(* CODESYS project slurryboss

Project tree, tasks and I/O mapping:
  CODESYS_Control_Win_V3_x64 : CODESYS Control Win V3 x64, CODESYS, version 3.5.20.0
    application Application
  CR1104 : ecomatDisplay43inch_64bit, ifm electronic, order no. 
      , version 3.5.19.4
    application Application
      libraries: ifmDevice_ecomatDisplay, * (ifm electronic); CmpBitmapPool, * (System); Util, 3.5.19.0 (System); Standard, 3.5.18.0 (System); SysTimer, * (System); BACnet2, 2.0.0.0 (CODESYS); CAA CiA 405, 4.1.0.0 (CAA Technical Workgroup); Element Collections, 3.5.17.0 (3S - Smart Software Solutions GmbH)
      task Task (cyclic, interval 1 ms, priority 0) calls PLC_PRG, Key_Lights, Test_PRG
      task VISU_TASK (cyclic, interval 10 ms, priority 15) calls VisuElems.Visu_Prg
      Components/
        KIQ Radar/
          function block fb_KIQ [LD]
          function block fbexample [LD]
        LMC500/
          data type eLMC500_State
          function block fb_LMC500 [LD]
        Purge/
          fb_Purge/
            data type ePurge_State
            function block fb_Purge [LD]: Volume_Calculation
            visualisation frame_PurgeStatus
        Slurry Pump/
          data type eSlurry_Pump_State
          function block fb_Slurry_Pump [LD]
        program Test_PRG [CFC]
        function block TOI [ST]
      Device/
        program Key_Lights [CFC]
      function block fb_KeyLight [ST]: Off, On, Set_Blue, Set_Green, Set_Previous, Set_Red, Set_White
      HMI/
        Components/
          Blind setting/
            visualisation f_BlindSetting
            function block fb_BlindSetting [LD]
          Buttons/
            visualisation f_Toggle_Button
          Checkbox/
            visualisation f_Checkbox
            function block fb_Checkbox [LD]
          Dial Indicator/
            visualisation f_DialIndicator
            function block fb_DialIndicator [ST]
          f_ProgressBar/
            visualisation f_ProgressBar
          global variables Global_Cards
          Menu/
            visualisation menu_demo
            image pool Menu_Images
            visualisation Menu_Item
            visualisation Right_Side_Nav
            function block swipe [LD]
          Pages/
            visualisation Analytics
            visualisation Chemistry
            visualisation Overview
            visualisation Pumps
            visualisation Purge
            visualisation Settings
          POUs/
            Hotkey/
              visualisation Tank_Frame
            function block Keypad_Navigation_FB [ST]: down, left, right, up
          interface selectable
          Setting Card/
            POUs/
              function block fb_Setting_Card [ST]: decrease, increase
            visualisation Test_Card
            Visus/
              visualisation Setting_Card_Frame
          visualisation Slurry_Pump_Card
      program PLC_PRG [CFC]
      global variables prvars
      program Test1 [CFC]
    Communication : Communication, ifm electronic, version 3.5.19.4
      CAN : CAN, ifm electronic, version 3.5.19.4
        CANbus_ecomatDisplay4_3 : CANbus_ecomatDisplay4.3, ifm electronic, version 1.0.0.0
          CANopen_Manager : CANopen_Manager, CODESYS, version 4.2.0.0
              settings: ConfigVersion = 50659584
            ODE3 : ODE3, Invertek Drives Ltd, order no. 0, version Revision=16#00000000, FileVersion=1.1, File=INVERTEK_ODE3_CANopen v3.00.eds
                settings: NODEIDSAVED = 1; SDO Timeout = 1000000; EXPERTSETTINGS = FALSE; Heartbeat-Producer Time = 200; Process by CANopenManager = TRUE; PDO 16#1401.COBID = 16#C0000301; Generic COBID = '$NODEID+16#C0000300'; Process by CANopenManager = TRUE; PDO 16#1800.Event Timer = 0; Process by CANopenManager = TRUE; PDO 16#1801.COBID = 16#C0000281; PDO 16#1801.Event Timer = 0; Generic COBID = '$NODEID+16#C0000280'; Process by CANopenManager = TRUE; Control Command Register.Subindex = 16#00; Speed Reference.Subindex = 16#00; User Ramp.Subindex = 16#00; no-name.Index = 16#0006; no-name.Subindex = 16#00; no-name.Index = 16#0006; no-name.Subindex = 16#00; no-name.Index = 16#0006; no-name.Subindex = 16#00; no-name.Index = 16#0006; no-name.Subindex = 16#00; no-name.Index = 16#0006; no-name.Subindex = 16#00; Drive Status Register.Subindex = 16#00; Motor Speed.Subindex = 16#00; Motor Current.Subindex = 16#00; Drive Temperature.Subindex = 16#00; DC Bus Voltage.Subindex = 16#00; Digital Input Status.Subindex = 16#00; Analog Input 1.Subindex = 16#00; Analog Input 2.Subindex = 16#00; SDO List.Set COB-ID sync.Index = 16#1005; SDO List.Set COB-ID sync.Subindex = 16#00; SDO List.Set COB-ID sync.Value = 16#00000080; SDO List.Set COB-ID sync.Size = 32; SDO List.Set COB-ID sync.AbortIfError = FALSE;
                  SDO List.Set COB-ID sync.JumpToLine = FALSE; SDO List.Set COB-ID sync.Line = 0; SDO List.Set Guardtime.Index = 16#100C; SDO List.Set Guardtime.Subindex = 16#00; SDO List.Set Guardtime.Value = 16#00000000; SDO List.Set Guardtime.Size = 16; SDO List.Set Guardtime.AbortIfError = FALSE; SDO List.Set Guardtime.JumpToLine = FALSE; SDO List.Set Guardtime.Line = 0; SDO List.Set Lifetime.Index = 16#100D; SDO List.Set Lifetime.Subindex = 16#00; SDO List.Set Lifetime.Value = 16#00000000; SDO List.Set Lifetime.Size = 8; SDO List.Set Lifetime.AbortIfError = FALSE; SDO List.Set Lifetime.JumpToLine = FALSE; SDO List.Set Lifetime.Line = 0; SDO List.Disable Emcy CobID.Index = 16#1014; SDO List.Disable Emcy CobID.Subindex = 16#00; SDO List.Disable Emcy CobID.Value = 16#80000081; SDO List.Disable Emcy CobID.Size = 32; SDO List.Disable Emcy CobID.AbortIfError = FALSE; SDO List.Disable Emcy CobID.JumpToLine = FALSE; SDO List.Disable Emcy CobID.Line = 0; SDO List.Set Emcy CobID.Index = 16#1014; SDO List.Set Emcy CobID.Subindex = 16#00; SDO List.Set Emcy CobID.Value = 16#00000081; SDO List.Set Emcy CobID.Size = 32; SDO List.Set Emcy CobID.AbortIfError = FALSE; SDO List.Set Emcy CobID.JumpToLine = FALSE; SDO List.Set Emcy CobID.Line = 0; SDO List.Set Heartbeat Producer.Index = 16#1017; SDO List.Set Heartbeat Producer.Subindex = 16#00; SDO List.Set Heartbeat Producer.Value = 16#000000C8; SDO List.Set Heartbeat Producer.Size = 16; SDO List.Set Heartbeat Producer.AbortIfError = FALSE; SDO List.Set Heartbeat Producer.JumpToLine = FALSE; SDO List.Set Heartbeat Producer.Line = 0; SDO List.Disable PDO.Index = 16#1400; SDO List.Disable PDO.Subindex = 16#01; SDO List.Disable PDO.Value = 16#C0000201;
                  SDO List.Disable PDO.Size = 32; SDO List.Disable PDO.AbortIfError = FALSE; SDO List.Disable PDO.JumpToLine = FALSE; SDO List.Disable PDO.Line = 0; SDO List.Set transmission type.Index = 16#1400; SDO List.Set transmission type.Subindex = 16#02; SDO List.Set transmission type.Value = 16#FE; SDO List.Set transmission type.Size = 8; SDO List.Set transmission type.AbortIfError = FALSE; SDO List.Set transmission type.JumpToLine = FALSE; SDO List.Set transmission type.Line = 0; SDO List.Clear pdo mapping.Index = 16#1600; SDO List.Clear pdo mapping.Subindex = 16#00; SDO List.Clear pdo mapping.Value = 16#0; SDO List.Clear pdo mapping.Size = 8; SDO List.Clear pdo mapping.AbortIfError = FALSE; SDO List.Clear pdo mapping.JumpToLine = FALSE; SDO List.Clear pdo mapping.Line = 0; SDO List.Set Mapping.Index = 16#1600; SDO List.Set Mapping.Subindex = 16#01; SDO List.Set Mapping.Value = 16#20000010; SDO List.Set Mapping.Size = 32; SDO List.Set Mapping.AbortIfError = FALSE; SDO List.Set Mapping.JumpToLine = FALSE; SDO List.Set Mapping.Line = 0; SDO List.Set Mapping.Index = 16#1600; SDO List.Set Mapping.Subindex = 16#02; SDO List.Set Mapping.Value = 16#20010010; SDO List.Set Mapping.Size = 32; SDO List.Set Mapping.AbortIfError = FALSE; SDO List.Set Mapping.JumpToLine = FALSE; SDO List.Set Mapping.Line = 0; SDO List.Set Mapping.Index = 16#1600; SDO List.Set Mapping.Subindex = 16#03; SDO List.Set Mapping.Value = 16#20030010; SDO List.Set Mapping.Size = 32; SDO List.Set Mapping.AbortIfError = FALSE; SDO List.Set Mapping.JumpToLine = FALSE; SDO List.Set Mapping.Line = 0; SDO List.Set Mapping.Index = 16#1600;
                  SDO List.Set Mapping.Subindex = 16#04; SDO List.Set Mapping.Value = 16#00060010; SDO List.Set Mapping.Size = 32; SDO List.Set Mapping.AbortIfError = FALSE; SDO List.Set Mapping.JumpToLine = FALSE; SDO List.Set Mapping.Line = 0; SDO List.Set number of mappings.Index = 16#1600; SDO List.Set number of mappings.Subindex = 16#00; SDO List.Set number of mappings.Value = 16#04; SDO List.Set number of mappings.Size = 8; SDO List.Set number of mappings.AbortIfError = FALSE; SDO List.Set number of mappings.JumpToLine = FALSE; SDO List.Set number of mappings.Line = 0; SDO List.Set and enable COB-ID.Index = 16#1400; SDO List.Set and enable COB-ID.Subindex = 16#01; SDO List.Set and enable COB-ID.Value = 16#40000201; SDO List.Set and enable COB-ID.Size = 32; SDO List.Set and enable COB-ID.AbortIfError = FALSE; SDO List.Set and enable COB-ID.JumpToLine = FALSE; SDO List.Set and enable COB-ID.Line = 0; SDO List.Disable PDO.Index = 16#1401; SDO List.Disable PDO.Subindex = 16#01; SDO List.Disable PDO.Value = 16#C0000301; SDO List.Disable PDO.Size = 32; SDO List.Disable PDO.AbortIfError = FALSE; SDO List.Disable PDO.JumpToLine = FALSE; SDO List.Disable PDO.Line = 0; SDO List.Disable PDO.Index = 16#1800; SDO List.Disable PDO.Subindex = 16#01; SDO List.Disable PDO.Value = 16#C0000181; SDO List.Disable PDO.Size = 32; SDO List.Disable PDO.AbortIfError = FALSE; SDO List.Disable PDO.JumpToLine = FALSE; SDO List.Disable PDO.Line = 0; SDO List.Set transmission type.Index = 16#1800; SDO List.Set transmission type.Subindex = 16#02; SDO List.Set transmission type.Value = 16#FE; SDO List.Set transmission type.Size = 8; SDO List.Set transmission type.AbortIfError = FALSE; SDO List.Set transmission type.JumpToLine = FALSE;
                  SDO List.Set transmission type.Line = 0; SDO List.Set inhibit time.Index = 16#1800; SDO List.Set inhibit time.Subindex = 16#03; SDO List.Set inhibit time.Value = 16#0000; SDO List.Set inhibit time.Size = 16; SDO List.Set inhibit time.AbortIfError = FALSE; SDO List.Set inhibit time.JumpToLine = FALSE; SDO List.Set inhibit time.Line = 0; SDO List.Clear pdo mapping.Index = 16#1A00; SDO List.Clear pdo mapping.Subindex = 16#00; SDO List.Clear pdo mapping.Value = 16#0; SDO List.Clear pdo mapping.Size = 8; SDO List.Clear pdo mapping.AbortIfError = FALSE; SDO List.Clear pdo mapping.JumpToLine = FALSE; SDO List.Clear pdo mapping.Line = 0; SDO List.Set Mapping.Index = 16#1A00; SDO List.Set Mapping.Subindex = 16#01; SDO List.Set Mapping.Value = 16#200A0010; SDO List.Set Mapping.Size = 32; SDO List.Set Mapping.AbortIfError = FALSE; SDO List.Set Mapping.JumpToLine = FALSE; SDO List.Set Mapping.Line = 0; SDO List.Set Mapping.Index = 16#1A00; SDO List.Set Mapping.Subindex = 16#02; SDO List.Set Mapping.Value = 16#200B0010; SDO List.Set Mapping.Size = 32; SDO List.Set Mapping.AbortIfError = FALSE; SDO List.Set Mapping.JumpToLine = FALSE; SDO List.Set Mapping.Line = 0; SDO List.Set Mapping.Index = 16#1A00; SDO List.Set Mapping.Subindex = 16#03; SDO List.Set Mapping.Value = 16#200D0010; SDO List.Set Mapping.Size = 32; SDO List.Set Mapping.AbortIfError = FALSE; SDO List.Set Mapping.JumpToLine = FALSE; SDO List.Set Mapping.Line = 0; SDO List.Set Mapping.Index = 16#1A00; SDO List.Set Mapping.Subindex = 16#04; SDO List.Set Mapping.Value = 16#20100010; SDO List.Set Mapping.Size = 32;
                  SDO List.Set Mapping.AbortIfError = FALSE; SDO List.Set Mapping.JumpToLine = FALSE; SDO List.Set Mapping.Line = 0; SDO List.Set number of mappings.Index = 16#1A00; SDO List.Set number of mappings.Subindex = 16#00; SDO List.Set number of mappings.Value = 16#04; SDO List.Set number of mappings.Size = 8; SDO List.Set number of mappings.AbortIfError = FALSE; SDO List.Set number of mappings.JumpToLine = FALSE; SDO List.Set number of mappings.Line = 0; SDO List.Set and enable COB-ID.Index = 16#1800; SDO List.Set and enable COB-ID.Subindex = 16#01; SDO List.Set and enable COB-ID.Value = 16#40000181; SDO List.Set and enable COB-ID.Size = 32; SDO List.Set and enable COB-ID.AbortIfError = FALSE; SDO List.Set and enable COB-ID.JumpToLine = FALSE; SDO List.Set and enable COB-ID.Line = 0; SDO List.Disable PDO.Index = 16#1801; SDO List.Disable PDO.Subindex = 16#01; SDO List.Disable PDO.Value = 16#C0000281; SDO List.Disable PDO.Size = 32; SDO List.Disable PDO.AbortIfError = FALSE; SDO List.Disable PDO.JumpToLine = FALSE; SDO List.Disable PDO.Line = 0; ConfigVersion = 50659584
                unmapped channels: Control Command Register, Speed Reference, User Ramp, no-name, Drive Status Register, Motor Speed, Motor Current, Drive Temperature
      Ethernet : Ethernet, ifm electronic, version 3.5.19.4
  5ce3da45-db07-42e7-a21c-a00fff4ed8f6|C:\Users\johnm\Downloads\Full-Circle-Icon.png
  5ce3da45-db07-42e7-a21c-a00fff4ed8f6|C:\Users\johnm\Pictures\analytics icon.png
  5ce3da45-db07-42e7-a21c-a00fff4ed8f6|C:\Users\johnm\Pictures\demo branding button.png
  5ce3da45-db07-42e7-a21c-a00fff4ed8f6|C:\Users\johnm\Pictures\pump_3815797.png
  5ce3da45-db07-42e7-a21c-a00fff4ed8f6|C:\Users\johnm\Pictures\pump inverted.png
  text list GlobalTextList
*)

// CR1104/Application/Components/LMC500/eLMC500_State
{attribute 'qualified_only'}
{attribute 'strict'}
TYPE eLMC500_State :
(
	Disconnected := 0,
	Faulted:= 10,
	No_Detection:= 20,
	Water_Detected:= 30
);
END_TYPE

// CR1104/Application/Components/Slurry Pump/eSlurry_Pump_State
{attribute 'strict'}
{attribute 'to_string'}
TYPE eSlurry_Pump_State :
(
	Off := 0, //initial pseudo-state
	Disabled:= 10,
	Stopped_HL:= 20,
	Stopped_LL:= 25,
	Standby:= 30,
	Running:= 40
);
END_TYPE

// CR1104/Application/Components/Purge/fb_Purge/ePurge_State

{attribute 'strict'}
{attribute 'to_string'}
TYPE ePurge_State :
(
	Off := 0, //initial pseudo-state. No state displayed
	Disabled:= 10, //disabled by operator
	Standby:= 20, //enabled, not purging
	Purging:= 30 //purging
);
END_TYPE

// CR1104/Application/prvars
{attribute 'qualified_only'}
VAR_GLOBAL PERSISTENT RETAIN
	purge_frequency: UINT; //purge after x gallons
	purge_duration: UINT;
	purge_enabled: BOOL;
	slurry_pump_enabled: BOOL;
END_VAR

// CR1104/Application/HMI/Components/Global_Cards
{attribute 'qualified_only'}
VAR_GLOBAL
	Test_Navigation_Selection: ARRAY [0..4, 0..4] OF BOOL;;
END_VAR

// CR1104/Application/PLC_PRG
PROGRAM PLC_PRG
VAR
	setkeys: ifmDevice.ResetKeyMapping;
	setleds: ifmDevice.SetKeyLED; 
	Brightness: UDINT:= 16#00999999;
END_VAR

setkeys(xExecute := TRUE); // ifmDevice.ResetKeyMapping
setleds(xEnable := TRUE, udiColour := Brightness); // ifmDevice.SetKeyLED

END_PROGRAM

// CR1104/Application/Device/Key_Lights
PROGRAM Key_Lights
VAR_INPUT
	Brightness: REAL:= 1;
END_VAR
VAR
	KL: ARRAY [0..5] OF fb_KeyLight;
	setleds: ifmDevice.SetKeyLED; 
	//LED: ifmDevice.ControlAllKeyLEDs;

END_VAR

(*
4 -> 0
2 -> 1
0 -> 2
5 -> 3
3 -> 4
1 -> 5
*)

KL[2](Brightness_Setting := Brightness); // fb_KeyLight
KL[3](Brightness_Setting := Brightness); // fb_KeyLight
KL[1](Brightness_Setting := Brightness); // fb_KeyLight
KL[4](Brightness_Setting := Brightness); // fb_KeyLight
KL[0](Brightness_Setting := Brightness); // fb_KeyLight
KL[5](Brightness_Setting := Brightness); // fb_KeyLight
setleds(
    xEnable := NOT(setleds.xError),
    eLED_ID := ifmDevice.eKEY_LED_ID.KEY2_NAVIGATION,
    udiColour := KL[2].Color); // ifmDevice.SetKeyLED

END_PROGRAM

// CR1104/Application/fb_KeyLight
FUNCTION_BLOCK fb_KeyLight
VAR_INPUT
	Brightness_Setting: REAL:= 1; //0..1 real factor
END_VAR
VAR_OUTPUT
	Color: UDINT;
END_VAR
VAR
//	LED: ifmDevice.keyled;
	Red: REAL;
	Green: REAL;
	Blue: REAL;
	Light: REAL;
	Color_Memory: ARRAY [0..1] OF UDINT;
END_VAR

Color:=(
	SHL(TO_UDINT(Red * Light),16) + 	//16#00FF0000 values
	SHL(TO_UDINT(Green * Light),8) + 	//16#0000FF00 values
	TO_UDINT(Blue * Light)				//16#000000FF
);

IF Color_Memory[1] <> Color THEN
	Color_Memory[0]:= Color_Memory[1];
	Color_Memory[1]:= Color;
END_IF

METHOD Off
VAR_INPUT
END_VAR
THIS^.Light:= 0;
END_METHOD

METHOD On
VAR_INPUT
END_VAR
THIS^.Light:= THIS^.Brightness_Setting;
END_METHOD

METHOD Set_Blue
VAR_INPUT
END_VAR
THIS^.Red:= 0;
THIS^.Green:= 0;
THIS^.Blue:= 255;
END_METHOD

METHOD Set_Green
VAR_INPUT
END_VAR
END_METHOD

METHOD Set_Previous
VAR_INPUT
END_VAR
Red:= 	TO_REAL(16#00FF0000 AND Color_Memory[0]);
Green:= TO_REAL(16#0000FF00 AND Color_Memory[0]);
Blue:= 	TO_REAL(16#000000FF AND Color_Memory[0]);
END_METHOD

METHOD Set_Red
VAR_INPUT
END_VAR
END_METHOD

METHOD Set_White
VAR_INPUT
END_VAR
THIS^.Red:= 255;
THIS^.Green:= 255;
THIS^.Blue:= 255;
END_METHOD

END_FUNCTION_BLOCK

// CR1104/Application/Components/Test_PRG
PROGRAM Test_PRG
/////
VAR
	Purge_Control: fb_Purge;
	Slurry_Pump_Control: fb_Slurry_Pump;
	Slurry_Sensor: fb_LMC500;
	placeholder: ifmDevice.stKEY_MAP_LIST:= (eKey2_Return:= ifmDevice.eKey_Map_Codes.END);
	test_bit: BOOL;
END_VAR
/////
VAR
	Simu_Sys_On: BOOL;
	Simu_Pump_State: eSlurry_Pump_State;
	Simu_Tank_Level: UINT; 
	Simu_Sensor: eLMC500_State:= eLMC500_State.Water_Detected;
	keymap: ifmdevice.GetKeyMapping;
	set_map: ifmdevice.SetKeyMapping;
	test_toggle: fb_Checkbox;
	menu_swipe: swipe;
	Swipe_menu: BOOL;
END_VAR
/////

Slurry_Pump_Control(
    System_On := TRUE,
    Enabled := prvars.slurry_pump_enabled,
    Sensor := simu_sensor,
    Tank_Level := Simu_Tank_Level,
    Delay_Time := T#20s); // fb_Slurry_Pump
Purge_Control(
    System_On := TRUE,
    Enabled := prvars.purge_enabled,
    Pump_State := Slurry_Pump_Control.State,
    Gallons_Setpoint := prvars.purge_frequency,
    Purge_Duration := TO_TIME(prvars.purge_duration * 1000)); // fb_Purge
keymap(xExecute := NOT(keymap.xDone) AND NOT(keymap.xDone)); // ifmdevice.GetKeyMapping
set_map(xExecute := NOT(set_map.xDone OR set_map.xError), stKeyMapList := placeholder); // ifmdevice.SetKeyMapping
// parameter Slurry_Sensor.No_Detection_Value := 80
// parameter Slurry_Sensor.Detection_Value := 60
Slurry_Sensor(); // fb_LMC500
test_toggle(on := prvars.purge_enabled); // fb_Checkbox
// parameter menu_swipe.delay := T#1ms
// parameter menu_swipe.distance := 126
menu_swipe(on := Swipe_menu); // swipe
// TO_UINT(TO_REAL((Test_PRG.Purge_Control.Cycle_Volume) / TO_REAL(Test_PRG.Purge_Control.Gallons_Setpoint)) * 100): input not connected

END_PROGRAM

// CR1104/Application/Components/Purge/fb_Purge/fb_Purge
FUNCTION_BLOCK fb_Purge
VAR_INPUT
	System_On: BOOL;
	Enabled: BOOL;
	Hand_Purge: BOOL;
	Pump_State: eSlurry_Pump_State;
	Gallons_Setpoint: UINT; //how many gallons from ref_Slurry_Pump before purging
	Purge_Duration: TIME;
END_VAR
VAR_INPUT CONSTANT
	Time_To_Gallons: UINT:= 666; //ms per gallon
END_VAR
VAR_OUTPUT
	State: ePurge_State;
	Cycle_Volume: UINT;
END_VAR
VAR
	tmr_purge: TON;
	Cycle_Timer: TOI;
	ft_purge: F_TRIG;
END_VAR
VAR // added by the converter: edge detectors and wires of the graphical bodies
    _w1, _w2, _w3, _w4, _w5 : BOOL;
END_VAR

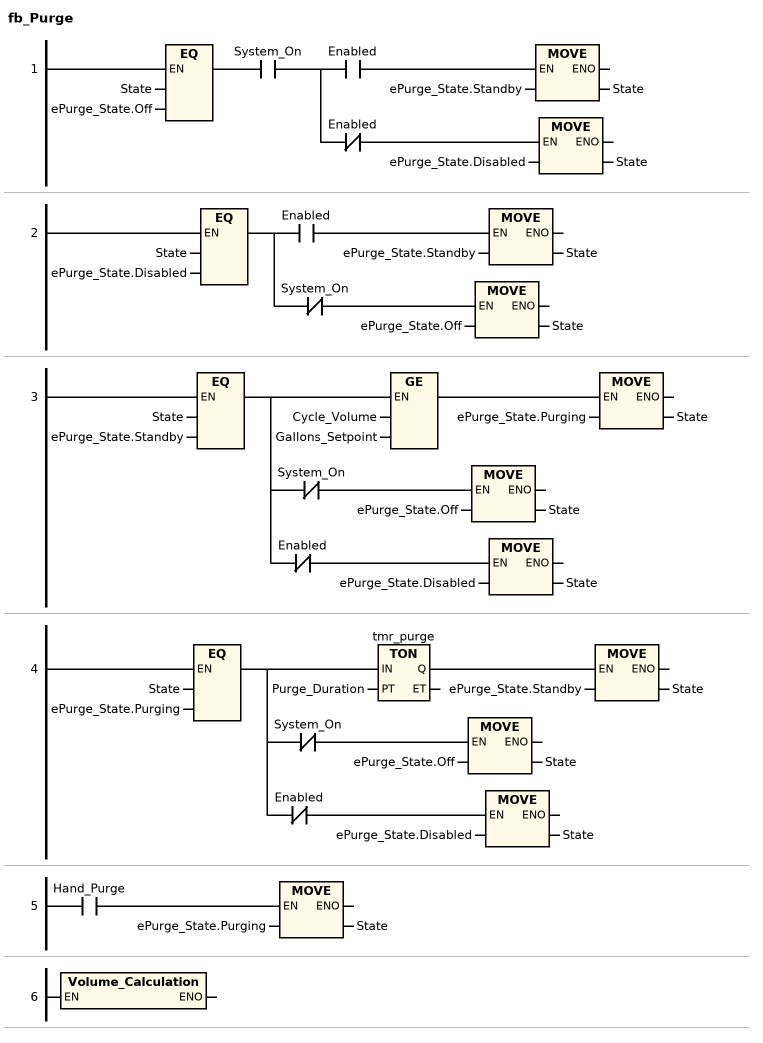
// NETWORK 1
_w1 := State = ePurge_State.Off AND System_On;
IF _w1 AND Enabled THEN State := ePurge_State.Standby; END_IF
IF _w1 AND NOT Enabled THEN State := ePurge_State.Disabled; END_IF

// NETWORK 2
_w2 := State = ePurge_State.Disabled;
IF _w2 AND Enabled THEN State := ePurge_State.Standby; END_IF
IF _w2 AND NOT System_On THEN State := ePurge_State.Off; END_IF

// NETWORK 3
_w3 := State = ePurge_State.Standby;
IF _w3 AND Cycle_Volume >= Gallons_Setpoint THEN State := ePurge_State.Purging; END_IF
IF _w3 AND NOT System_On THEN State := ePurge_State.Off; END_IF
IF _w3 AND NOT Enabled THEN State := ePurge_State.Disabled; END_IF

// NETWORK 4
_w4 := State = ePurge_State.Purging;
tmr_purge(IN := _w4, PT := Purge_Duration); // TON
IF tmr_purge.Q THEN State := ePurge_State.Standby; END_IF
IF _w4 AND NOT System_On THEN State := ePurge_State.Off; END_IF
IF _w4 AND NOT Enabled THEN State := ePurge_State.Disabled; END_IF

// NETWORK 5
IF Hand_Purge THEN State := ePurge_State.Purging; END_IF

// NETWORK 6
Volume_Calculation();

ACTION Volume_Calculation:
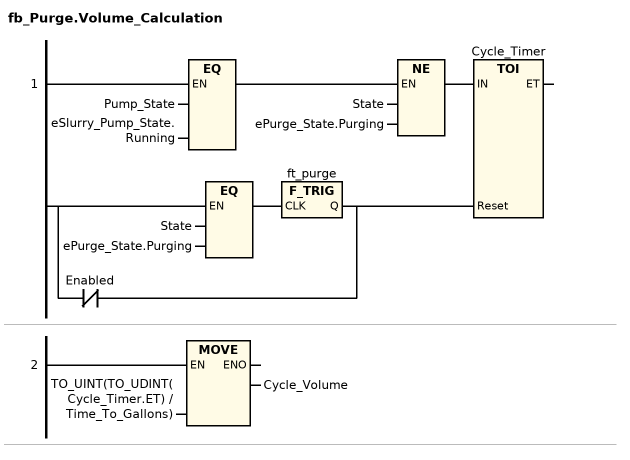
// NETWORK 1
_w5 := NOT Enabled;
IF NOT _w5 THEN
    ft_purge(CLK := State = ePurge_State.Purging); // F_TRIG
    _w5 := ft_purge.Q;
END_IF
Cycle_Timer(IN := Pump_State = eSlurry_Pump_State.Running AND State <> ePurge_State.Purging, Reset := _w5); // TOI

// NETWORK 2
Cycle_Volume := TO_UINT(TO_UDINT(Cycle_Timer.ET) / Time_To_Gallons);
END_ACTION

END_FUNCTION_BLOCK

// CR1104/Application/Components/TOI
FUNCTION_BLOCK TOI
VAR_INPUT
	IN : BOOL;
	Reset : BOOL;
END_VAR
VAR 
	TimerAdd: TIME; 
	CountingTimer: TIME;
	Trig: BOOL; 
	History: BOOL; 
	Pulse: BOOL; 
	TimerReset: BOOL; 
	Run: BOOL; 
	Running: BOOL; 
	StartTime: TIME;
	ResetONS: R_TRIG;
 END_VAR
 VAR_OUTPUT
	ET: TIME;
 END_VAR

ET:= TimerAdd + CountingTimer;
IF NOT IN THEN 
	IF Trig AND NOT History THEN 
		Pulse:= 1; History:= 1; Trig:= 0;
		ELSE 
			Pulse:= 0; History:= 1;
	END_IF
	IF Pulse THEN 
		CountingTimer:= ET;
	END_IF
	TimerReset:= 1;
END_IF
IF IN THEN 
	TimerReset:= 0;
	Trig:= 1; History:= 00;
END_IF
IF Reset THEN 
	TimerReset:= 1;
	CountingTimer:= T#001MS;
	ET:= T#001MS;
END_IF

Run:= NOT(TimerReset);

IF Run AND NOT Running THEN
	StartTime:= TIME();
	Running:= TRUE; END_IF
IF NOT Run AND NOT Running THEN
	StartTime:= TIME(); END_IF
ResetONS(clk:= TimerReset); 
IF ResetONS.Q THEN
	Running:= FALSE;
	StartTime:= TIME(); 
END_IF

TimerAdd:= TIME()-StartTime;

END_FUNCTION_BLOCK

// CR1104/Application/Components/Slurry Pump/fb_Slurry_Pump
FUNCTION_BLOCK fb_Slurry_Pump
VAR_INPUT
	System_On: BOOL;
	Enabled: BOOL;
	Sensor: eLMC500_State;
	Tank_Level: UINT;
	Delay_Time: TIME;
END_VAR
VAR_OUTPUT
	State: eSlurry_Pump_State;
END_VAR
VAR
	tmr_delay: TON;
	tmr_off: TON;
END_VAR
VAR // added by the converter: edge detectors and wires of the graphical bodies
    _w1, _w2, _w3, _w4, _w5 : BOOL;
END_VAR

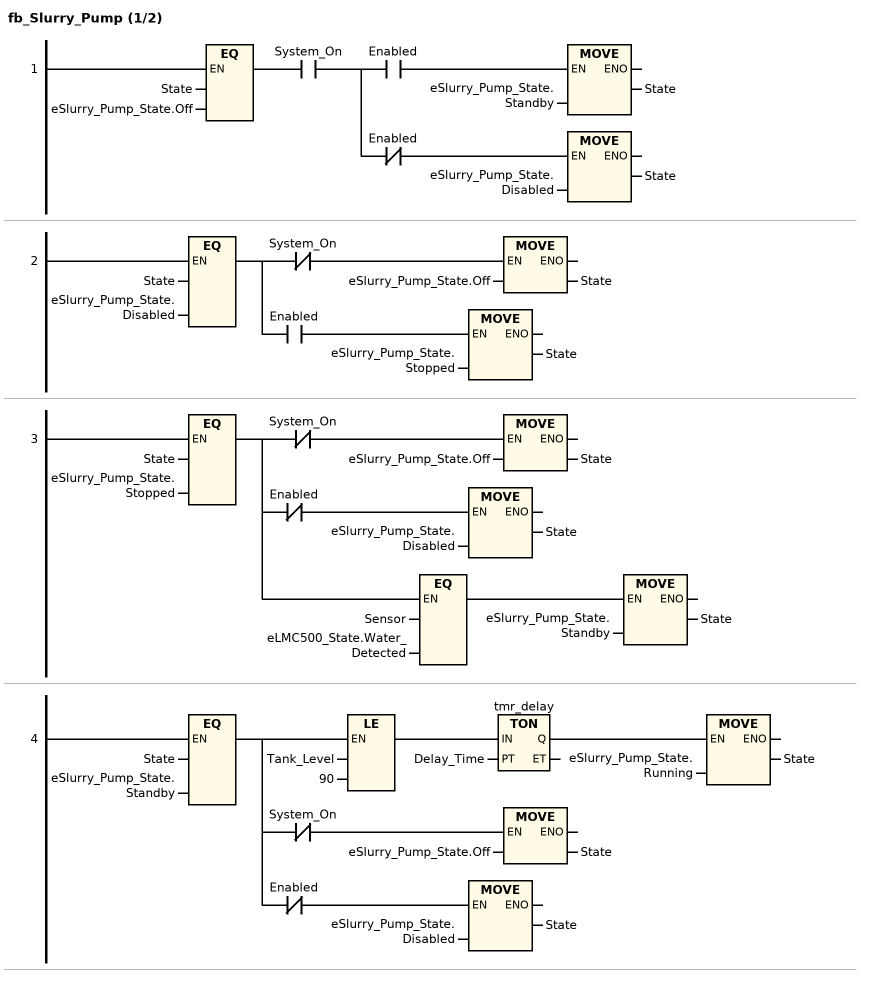
// NETWORK 1
_w1 := State = eSlurry_Pump_State.Off AND System_On;
IF _w1 AND Enabled THEN State := eSlurry_Pump_State.Standby; END_IF
IF _w1 AND NOT Enabled THEN State := eSlurry_Pump_State.Disabled; END_IF

// NETWORK 2
_w2 := State = eSlurry_Pump_State.Disabled;
IF _w2 AND NOT System_On THEN State := eSlurry_Pump_State.Off; END_IF
IF _w2 AND Enabled THEN State := eSlurry_Pump_State.Stopped; END_IF

// NETWORK 3
_w3 := State = eSlurry_Pump_State.Stopped;
IF _w3 AND NOT System_On THEN State := eSlurry_Pump_State.Off; END_IF
IF _w3 AND NOT Enabled THEN State := eSlurry_Pump_State.Disabled; END_IF
IF _w3 AND Sensor = eLMC500_State.Water_Detected THEN State := eSlurry_Pump_State.Standby; END_IF

// NETWORK 4
_w4 := State = eSlurry_Pump_State.Standby;
tmr_delay(IN := _w4 AND Tank_Level <= 90, PT := Delay_Time); // TON
IF tmr_delay.Q THEN State := eSlurry_Pump_State.Running; END_IF
IF _w4 AND NOT System_On THEN State := eSlurry_Pump_State.Off; END_IF
IF _w4 AND NOT Enabled THEN State := eSlurry_Pump_State.Disabled; END_IF

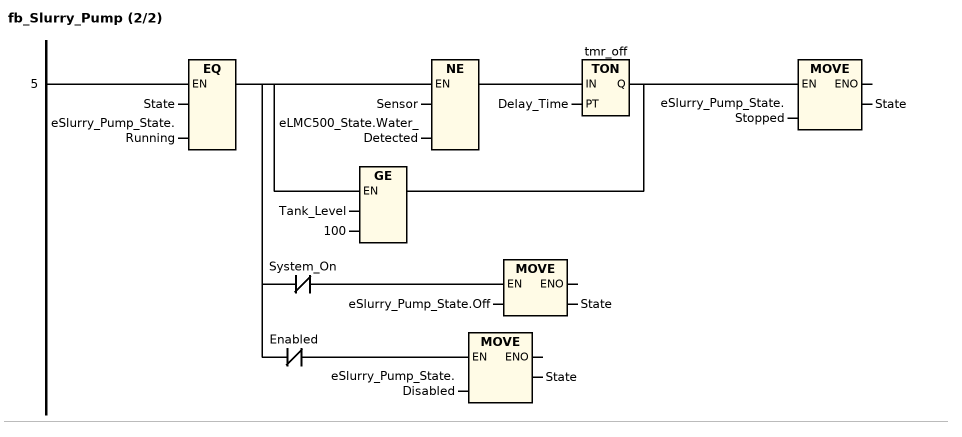
// NETWORK 5
_w5 := State = eSlurry_Pump_State.Running;
tmr_off(IN := _w5 AND Sensor <> eLMC500_State.Water_Detected, PT := Delay_Time); // TON
IF tmr_off.Q OR _w5 AND Tank_Level >= 100 THEN State := eSlurry_Pump_State.Stopped; END_IF
IF _w5 AND NOT System_On THEN State := eSlurry_Pump_State.Off; END_IF
IF _w5 AND NOT Enabled THEN State := eSlurry_Pump_State.Disabled; END_IF

END_FUNCTION_BLOCK

// CR1104/Application/Components/LMC500/fb_LMC500
FUNCTION_BLOCK fb_LMC500
/// 
VAR_INPUT
	IOL_Read: ARRAY [0..7] OF WORD;
END_VAR
///
VAR_OUTPUT
	state: eLMC500_State;
END_VAR
///
VAR_INPUT CONSTANT
	Detection_Value: UINT; //0-100
	No_Detection_Value: UINT; //0-100
END_VAR

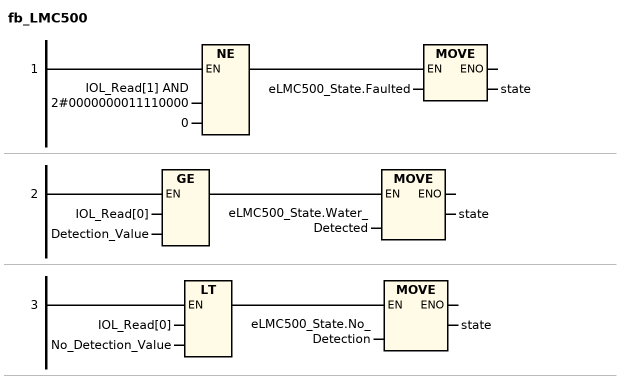
// NETWORK 1
IF (IOL_Read[1] AND 2#0000000011110000) <> 0 THEN state := eLMC500_State.Faulted; END_IF

// NETWORK 2
IF IOL_Read[0] >= Detection_Value THEN state := eLMC500_State.Water_Detected; END_IF

// NETWORK 3
IF IOL_Read[0] < No_Detection_Value THEN state := eLMC500_State.No_Detection; END_IF

END_FUNCTION_BLOCK

// CR1104/Application/HMI/Components/Checkbox/fb_Checkbox
FUNCTION_BLOCK fb_Checkbox
/////
VAR_IN_OUT
	on: BOOL;
END_VAR
/////
VAR_OUTPUT
	position: UINT;
END_VAR
////
VAR
	pos_ctu: CTU;
	pos_ctd: CTD;
	tmr_delay: TON;
	tmr_delay2: TON;
	off_trig: R_TRIG;
END_VAR
/////
VAR_INPUT CONSTANT
	delay: TIME:= T#2MS;
END_VAR
/////

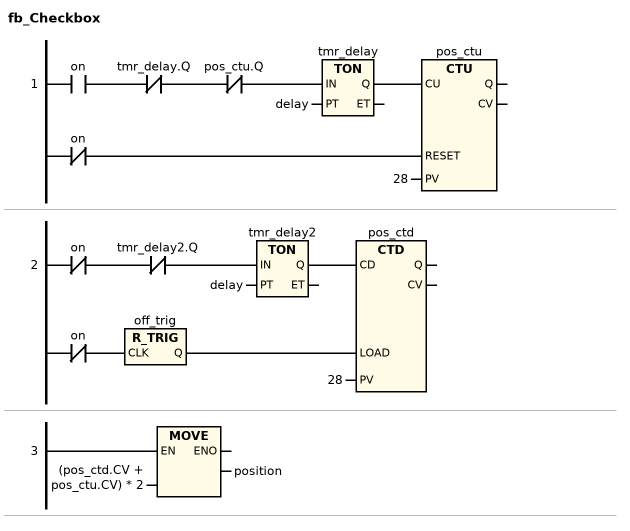
// NETWORK 1
tmr_delay(IN := on AND NOT tmr_delay.Q AND NOT pos_ctu.Q, PT := delay); // TON
pos_ctu(CU := tmr_delay.Q, RESET := NOT on, PV := 28); // CTU

// NETWORK 2
tmr_delay2(IN := NOT on AND NOT tmr_delay2.Q, PT := delay); // TON
off_trig(CLK := NOT on); // R_TRIG
pos_ctd(CD := tmr_delay2.Q, LOAD := off_trig.Q, PV := 28); // CTD

// NETWORK 3
position := (pos_ctd.CV + pos_ctu.CV) * 2;

END_FUNCTION_BLOCK

// CR1104/Application/HMI/Components/Menu/swipe
FUNCTION_BLOCK swipe
VAR_INPUT
	on: BOOL;
END_VAR
VAR_OUTPUT
	position: UINT;
END_VAR
VAR
	pos_ctu: CTU;
	pos_ctd: CTD;
	tmr_delay: TON;
	tmr_delay2: TON;
	off_trig: R_TRIG;
END_VAR
VAR_INPUT CONSTANT
	delay: TIME:= T#2MS;
	distance: UINT;
END_VAR

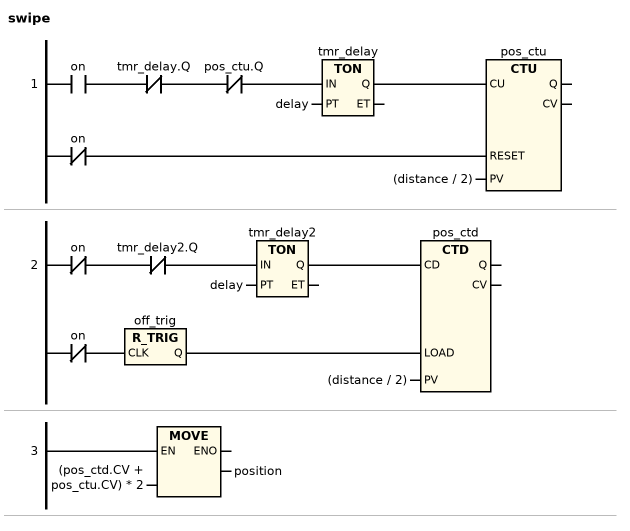
// NETWORK 1
tmr_delay(IN := on AND NOT tmr_delay.Q AND NOT pos_ctu.Q, PT := delay); // TON
pos_ctu(CU := tmr_delay.Q, RESET := NOT on, PV := (distance / 2)); // CTU

// NETWORK 2
tmr_delay2(IN := NOT on AND NOT tmr_delay2.Q, PT := delay); // TON
off_trig(CLK := NOT on); // R_TRIG
pos_ctd(CD := tmr_delay2.Q, LOAD := off_trig.Q, PV := (distance / 2)); // CTD

// NETWORK 3
position := (pos_ctd.CV + pos_ctu.CV) * 2;

END_FUNCTION_BLOCK

// CR1104/Application/Test1
PROGRAM Test1
VAR //test
END_VAR

END_PROGRAM

// CR1104/Application/Components/KIQ Radar/fb_KIQ
FUNCTION_BLOCK fb_KIQ
VAR_INPUT
END_VAR
VAR_OUTPUT
END_VAR
VAR
END_VAR

// NETWORK 1

END_FUNCTION_BLOCK

// CR1104/Application/Components/KIQ Radar/fbexample
FUNCTION_BLOCK fbexample
VAR_INPUT
END_VAR
VAR_OUTPUT
END_VAR
VAR
	active: BOOL;
	start_s2: BOOL;
	valve_q1: BOOL;
	highlevel_s5: BOOL;
	manual: BOOL;
	manual_mode: BOOL;
	manual_q1_button: BOOL;
END_VAR

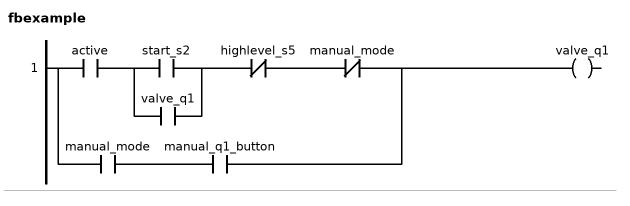
// NETWORK 1
valve_q1 := active AND (start_s2 OR valve_q1) AND NOT highlevel_s5 AND NOT manual_mode OR manual_mode AND manual_q1_button;

END_FUNCTION_BLOCK

// CR1104/Application/HMI/Components/selectable
INTERFACE selectable

END_INTERFACE

// CR1104/Application/HMI/Components/Blind setting/fb_BlindSetting
FUNCTION_BLOCK fb_BlindSetting
VAR_INPUT
	hover: BOOL;
	select: BOOL;
END_VAR
VAR_OUTPUT
	position: UINT;
END_VAR
VAR
	swipe_open: swipe;
END_VAR

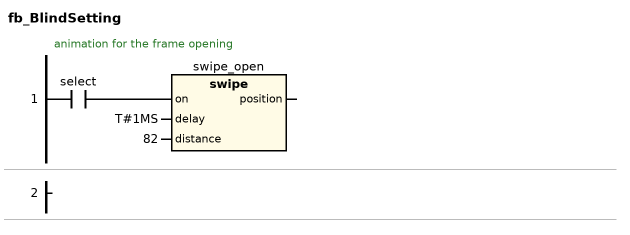
// NETWORK 1
// animation for the frame opening
swipe_open(on := select, delay := T#1MS, distance := 82); // swipe

// NETWORK 2

END_FUNCTION_BLOCK

// CR1104/Application/HMI/Components/Dial Indicator/fb_DialIndicator
FUNCTION_BLOCK fb_DialIndicator
VAR_INPUT
	r_Value: REFERENCE TO REAL;
	ui_Value: REFERENCE TO UINT;
	t_Value: REFERENCE TO TIME;
	Max_Value: UINT; //ms for time
	Name: STRING;
	Units: STRING;
END_VAR
VAR_OUTPUT
	Indicator_Val: UINT;
	xREAL: BOOL;
	xUINT: BOOL;
	xTIME: BOOL;
END_VAR
VAR
END_VAR


xREAL:= __ISVALIDREF(r_Value);
xUINT:= __ISVALIDREF(ui_Value);
xTIME:= __ISVALIDREF(t_Value);

IF xREAL THEN
	Indicator_Val:= 180 - TO_UINT((r_Value / TO_REAL(Max_Value)) * 180.0); //coefficient from proportion of max val
END_IF

END_FUNCTION_BLOCK

// CR1104/Application/HMI/Components/POUs/Keypad_Navigation_FB
FUNCTION_BLOCK Keypad_Navigation_FB
VAR_INPUT CONSTANT
	X_items: USINT; // How many items wide is the selection
	Y_items: USINT; // How many items tall is the selection
END_VAR
VAR_OUTPUT
	Position_X: USINT:= 0; //starting spot x
	Position_Y: USINT:= 0; //starting spot y
END_VAR

METHOD down
IF THIS^.Position_Y < THIS^.Y_items - 1 THEN
	THIS^.Position_Y:= THIS^.Position_Y + 1;
END_IF
END_METHOD

METHOD left
VAR_INPUT
END_VAR
IF THIS^.Position_X > 0 THEN
	THIS^.Position_X := THIS^.Position_X - 1;
END_IF
END_METHOD

METHOD right
VAR_INPUT
END_VAR
IF THIS^.Position_X < THIS^.X_Items - 1 THEN
	THIS^.Position_X := THIS^.Position_X + 1;
END_IF
END_METHOD

METHOD up
VAR_INPUT
END_VAR
IF THIS^.Position_Y > 0 THEN
	THIS^.Position_Y:= THIS^.Position_Y - 1;
END_IF
END_METHOD

END_FUNCTION_BLOCK

// CR1104/Application/HMI/Components/Setting Card/POUs/fb_Setting_Card
FUNCTION_BLOCK fb_Setting_Card
VAR_IN_OUT
	Value: UINT;
END_VAR
VAR_INPUT
	increment: UINT:= 1;
END_VAR
VAR_INPUT CONSTANT
	maximum: UINT;
	minimum: UINT;
END_VAR
VAR_OUTPUT
END_VAR
VAR
END_VAR

METHOD decrease
VAR_INPUT
END_VAR
IF THIS^.minimum >= THIS^.Value THEN
	RETURN;
END_IF

THIS^.Value:= THIS^.Value - increment;
END_METHOD

METHOD increase
VAR_INPUT
END_VAR
IF THIS^.maximum <= THIS^.Value THEN
	RETURN;
END_IF

THIS^.Value:= THIS^.Value + increment;
END_METHOD

END_FUNCTION_BLOCK

// CR1104/Application/HMI/Components/Slurry_Pump_Card
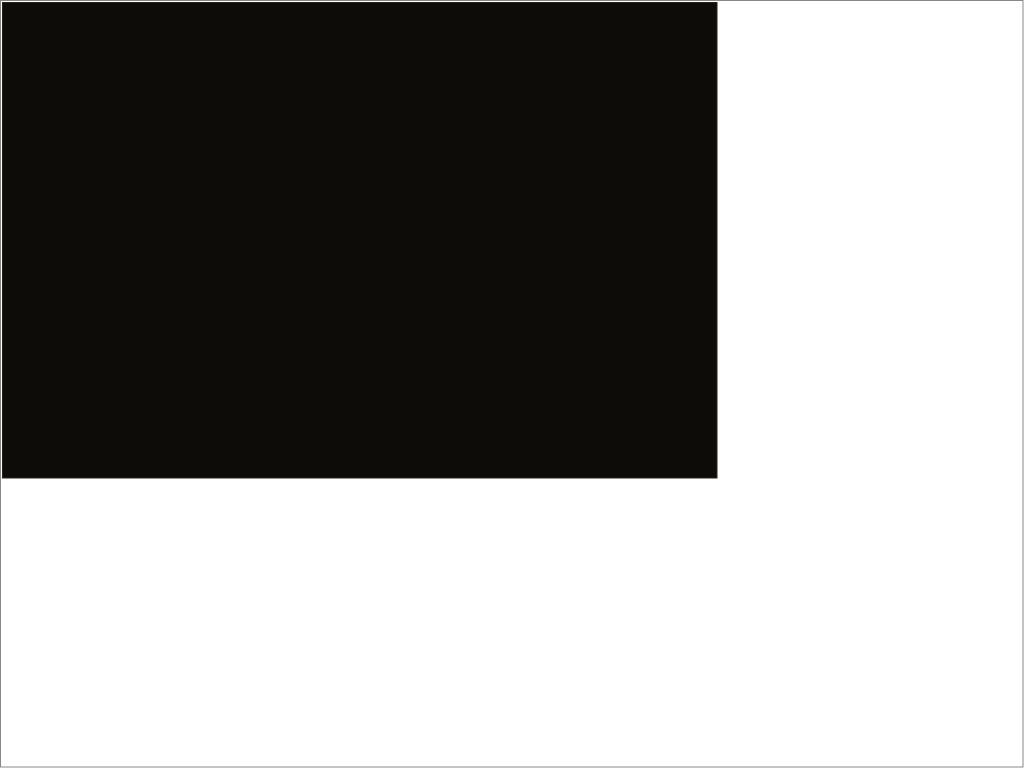
VISUALIZATION Slurry_Pump_Card  // 1024x768
VAR_INPUT
	_SELECTED: BOOL;
END_VAR
VAR
	Navigate: Keypad_Navigation_FB; 
END_VAR
    RoundedRectangle (2,2 715x476), colour toggle: _SELECTED
        p3560616238: TO_INT(_SELECTED) * (-116)
    hotkey  Id=481040531456, Key=KeyDown=True, KeyName=up, ActionToExecute=Action=STSnippet=IF NOT(_SELECTED) THEN RETURN; END_IF Navigate.up();, VisuElemId=-1
    hotkey  Id=481039482880, Key=KeyDown=True, KeyName=down, ActionToExecute=Action=STSnippet=IF NOT(_SELECTED) THEN RETURN; END_IF Navigate.down();, VisuElemId=-1
    hotkey  Id=481038434304, Key=KeyDown=True, KeyName=left, ActionToExecute=Action=STSnippet=IF NOT(_SELECTED) THEN RETURN; END_IF Navigate.left();, VisuElemId=-1
    hotkey  Id=481037385728, Key=KeyDown=True, KeyName=right, ActionToExecute=Action=STSnippet=IF NOT(_SELECTED) THEN RETURN; END_IF Navigate.right();, VisuElemId=-1
END_VISUALIZATION

// CR1104/Application/Components/Purge/fb_Purge/frame_PurgeStatus
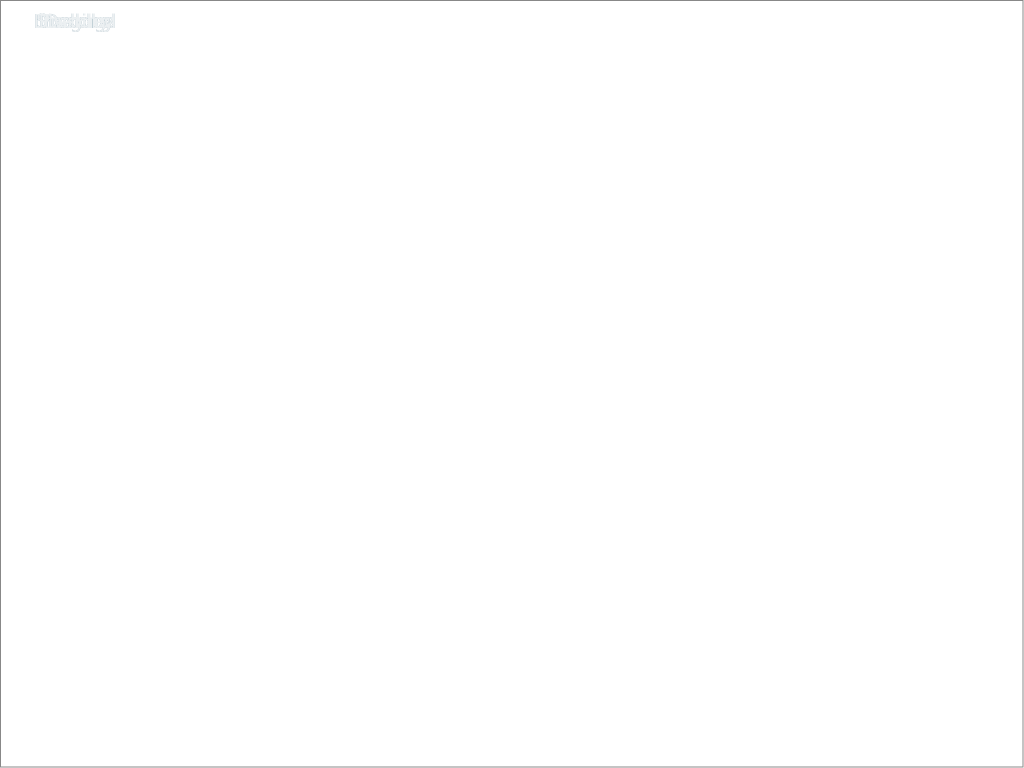
VISUALIZATION frame_PurgeStatus  // 1024x768
VAR_INPUT
	State: ePurge_State;
	Selected: BOOL;
END_VAR
    RoundedRectangle (0,0 150x43), "Debug", invisible if: State <> ePurge_State.Off
    RoundedRectangle (0,0 150x43), "Disabled", invisible if: State <> ePurge_State.Disabled
    RoundedRectangle (0,0 150x43), "Standby", invisible if: State <> ePurge_State.Standby
    RoundedRectangle (0,0 150x43), "Purging", invisible if: State <> ePurge_State.Purging
    RoundedRectangle (0,0 150x43), "Debug", invisible if: State <> ePurge_State.Off OR NOT(Selected)
    RoundedRectangle (0,0 150x43), "Disabled", invisible if: State <> ePurge_State.Disabled OR NOT(Selected)
    RoundedRectangle (0,0 150x43), "Standby", invisible if: State <> ePurge_State.Standby OR NOT(Selected)
    RoundedRectangle (0,0 150x43), "Purging", invisible if: State <> ePurge_State.Purging OR NOT(Selected)
END_VISUALIZATION

// CR1104/Application/HMI/Components/Blind setting/f_BlindSetting
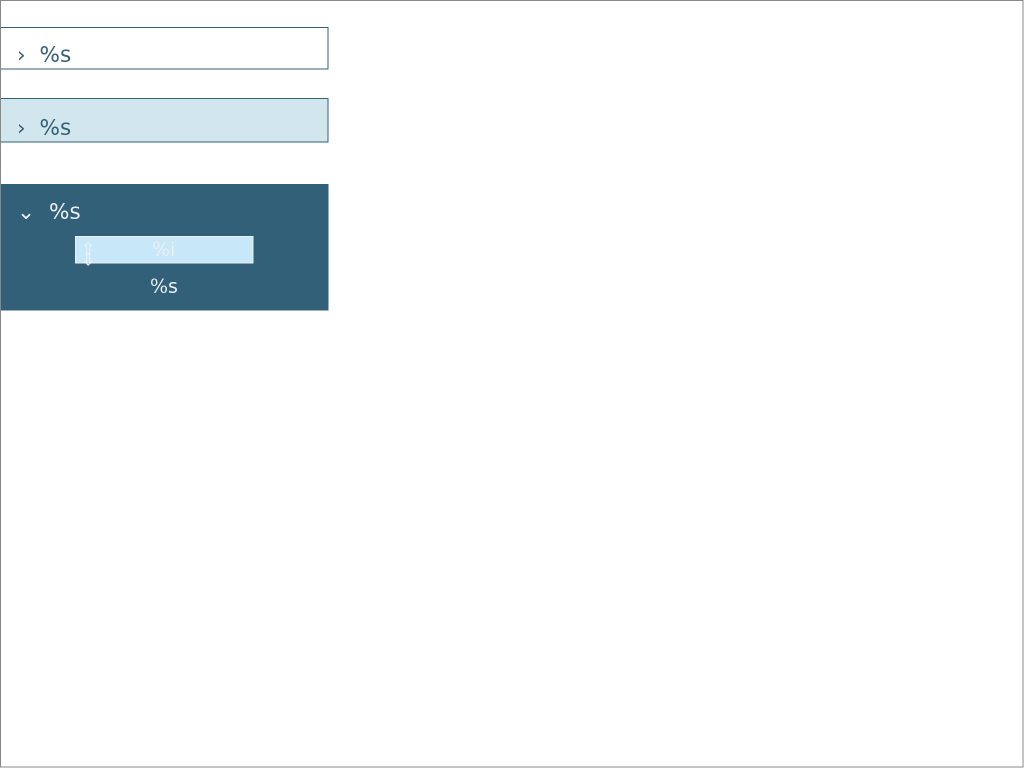
VISUALIZATION f_BlindSetting  // 1024x768
VAR_INPUT
	fb_ref: REFERENCE TO fb_BlindSetting;
END_VAR
    Rectangle (0,27 328x42), "› %s"
    Rectangle (0,184 328x126)
    RoundedRectangle (75,236 178x27), "%i"
    RoundedRectangle (0,264 328x27), "%s"
    Rectangle (0,184 328x42), "⌄ %s"
    RoundedRectangle (75,248 26x13), "⇩"
    RoundedRectangle (75,237 26x13), "⇧"
    Rectangle (0,98 328x44), invisible if: NOT(Hover)
    Rectangle (0,98 328x44), "› %s"
    RoundedRectangle (0,273 328x27), "%s"
END_VISUALIZATION

// CR1104/Application/HMI/Components/Buttons/f_Toggle_Button
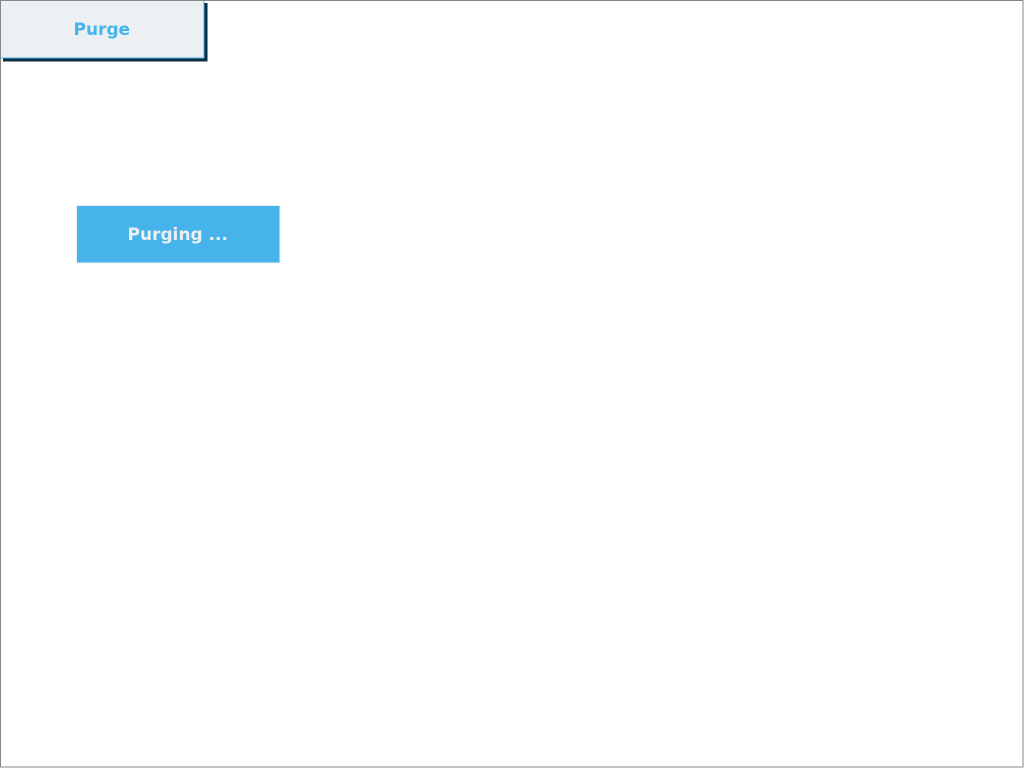
VISUALIZATION f_Toggle_Button  // 1024x768
    Rectangle (76,205 204x58)
    Rectangle (3,3 204x58)
    Rectangle (0,0 204x58), "Purge"
    Rectangle (76,205 204x58), "Purging ..."
END_VISUALIZATION

// CR1104/Application/HMI/Components/Checkbox/f_Checkbox
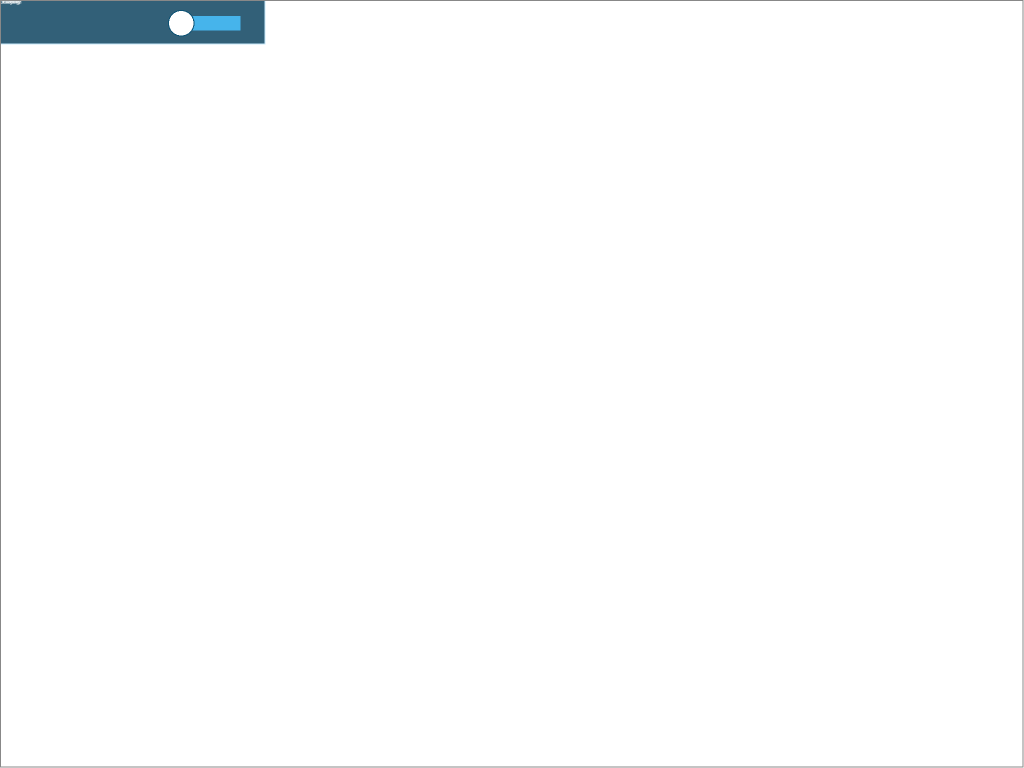
VISUALIZATION f_Checkbox  // 1024x768
VAR_IN_OUT
	Setting: BOOL;
END_VAR
VAR_INPUT
	fb_ref: REFERENCE TO fb_Checkbox;
	Name: STRING;
	Hover: BOOL;
	Selected: BOOL;
END_VAR
    Rectangle (0,0 265x44)
    Rectangle (0,0 265x44), invisible if: NOT(Hover)
    Rectangle (0,0 265x44), invisible if: NOT(Selected)
    Group (184,16 56x14)
        RoundedRectangle (0,0 56x14)
        RoundedRectangle (0,0 56x14), invisible if: NOT(fb_ref.on)
    Ellipse (168,10 26x26)
        p3560616238: fb_ref.position
    Frame (0,0 152x44)
        shows frame_PurgeStatus(State := Test_PRG.Purge_Control.State, Selected := Selected)
    hotkey  Id=481037385728, Key=KeyDown=True, KeyName=up, ActionToExecute=Action=STSnippet=IF NOT Selected THEN RETURN; END_IF fb_ref.on:= false;, VisuElemId=-1
    hotkey  Id=481038434304, Key=KeyName=down, ActionToExecute=Action=STSnippet=IF NOT Selected THEN RETURN; END_IF fb_ref.on:= TRUE;, VisuElemId=-1
END_VISUALIZATION

// CR1104/Application/HMI/Components/Dial Indicator/f_DialIndicator
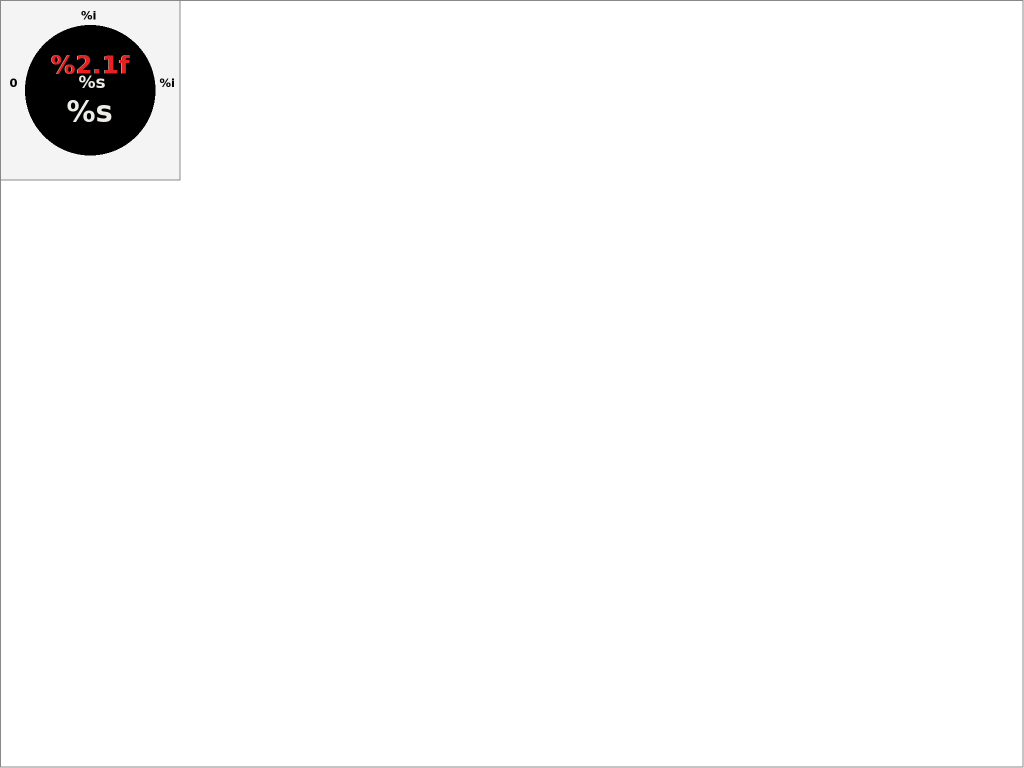
VISUALIZATION f_DialIndicator  // 1024x768
VAR_INPUT
	background: DWORD; 
	fb_Ref: fb_DialIndicator;
	Alarm: BOOL;
	layer: DWORD;
END_VAR
    Pie (0,0 180x180)
    Pie (0,0 180x180)
        p2124672552: fb_Ref.Indicator_Val
    Pie (0,0 180x180), invisible if: NOT(Alarm)
        p2124672552: fb_Ref.Indicator_Val
    Ellipse (25,25 130x130), colour variable: layer
        p3450524324: layer
    Group (0,0 180x98)
        Rectangle (155,68 25x30), "%i", text variable: fb_Ref.Max_Value
        Rectangle (67,0 44x31), "%i", text variable: TO_REAL(fb_Ref.Max_Value) * 0.5
        Rectangle (0,68 27x30), "0"
    RoundedRectangle (25,50 130x30), "%2.1f", text variable: fb_Ref.r_Value
    RoundedRectangle (36,50 109x30), "%2.1f", text variable: fb_Ref.r_Value, invisible if: NOT(Alarm)
    Rectangle (37,71 110x22), "%s", text variable: fb_Ref.Units
    Rectangle (0,90 180x43), "%s", text variable: fb_Ref.Name
END_VISUALIZATION

// CR1104/Application/HMI/Components/f_ProgressBar/f_ProgressBar
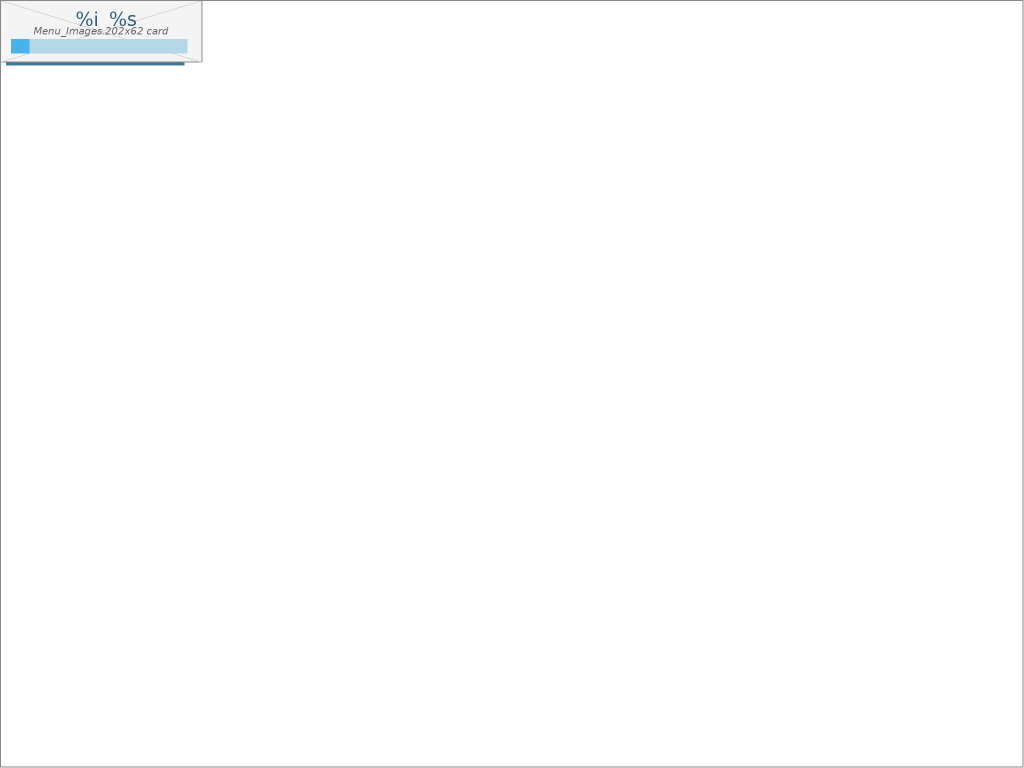
VISUALIZATION f_ProgressBar  // 1024x768
VAR_INPUT
	Value: UINT;
	Percentage: UINT; 
	Units: STRING;
END_VAR
    RoundedRectangle (6,5 178x60)
    Image (0,0 202x62), image: Menu_Images.202x62 card
    RoundedRectangle (11,39 176x14)
    RoundedRectangle (11,39 18x14)
        p874137650: TO_UINT(TO_REAL(Percentage) * 1.55)
    RoundedRectangle (16,5 86x29), "%i", text variable: Value
    RoundedRectangle (106,5 81x29), "%s", text variable: Units
END_VISUALIZATION

// CR1104/Application/HMI/Components/Menu/menu_demo
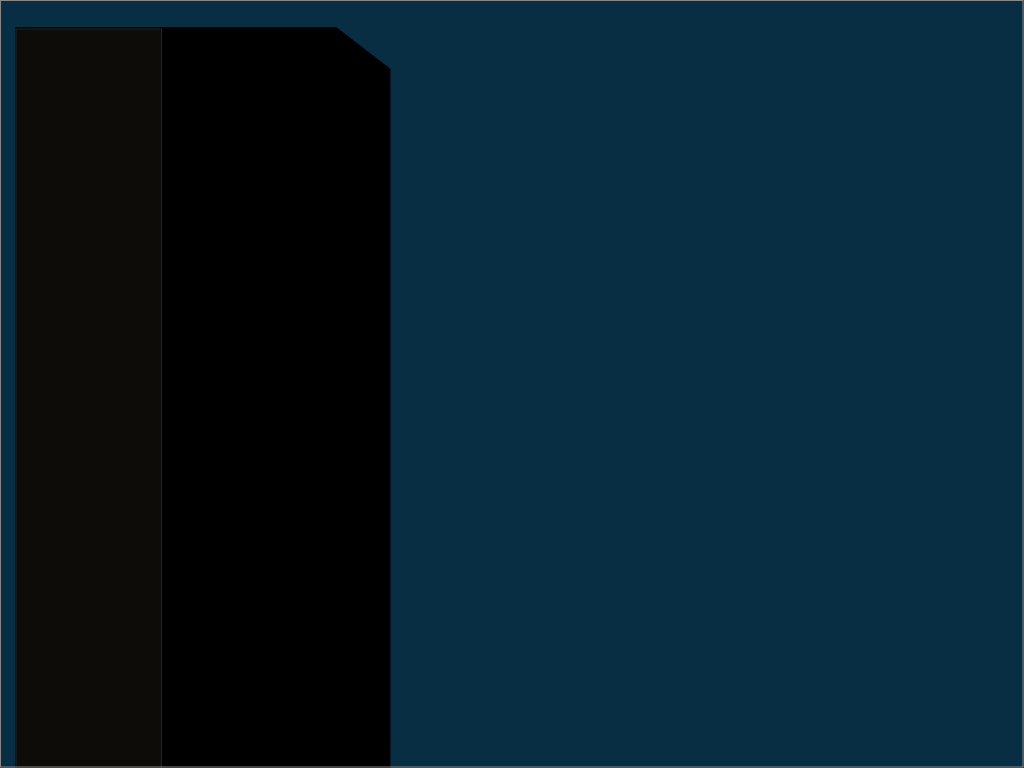
VISUALIZATION menu_demo  // 1024x768
VAR
	Show_Menu: BOOL;
	var1: UINT;
	var2: UINT;
	bool1: BOOL;
	
	Hover_X: UINT;
	Hover_Y: UINT;
	Selected: ARRAY [0..1, 0..5] OF BOOL;
	xSelected: BOOL;
	
	Visu_Index: UINT;
END_VAR
    Frame (14,0 575x762)
        shows Right_Side_Nav(Show_Menu := Test_PRG.Swipe_menu, Select_Y := Visu_Index)
        p3560616238: -1.0 * (Test_PRG.menu_swipe.position)
    Frame (15,27 375x741), frame switch variable: Visu_Index
        shows Overview()
        shows Pumps()
        shows Purge(xSELECTED := xSelected, Hover_X := Hover_X)
        shows Chemistry()
        shows Analytics()
        shows Settings()
        p2292087262: xSelected
        p384951027: Hover_Y
        p1643565669: Hover_X
        p3560616238: -1.0 * (Test_PRG.menu_swipe.position)
    Polygon (346,12) (366,2) (400,16) (391,69) (334,25)
        p3560616238: -1.0 * (Test_PRG.menu_swipe.position)
    hotkey  Id=481039482880, Key=KeyDown=True, KeyName=up, ActionToExecute=Action=STSnippet=IF xSelected THEN RETURN; END_IF IF Test_PRG.Swipe_menu = 1 THEN Test_PRG.Swipe_menu:= 0; END_IF, VisuElemId=-1
    hotkey  Id=481040531456, Key=KeyDown=True, KeyName=down, ActionToExecute=Action=STSnippet=IF xSelected THEN RETURN; END_IF IF Test_PRG.Swipe_menu = 0 THEN Test_PRG.Swipe_menu:= 1; END_IF, VisuElemId=-1
    hotkey  Id=481042628608, Key=KeyDown=True, KeyName=left, ActionToExecute=Action=STSnippet=IF xSelected THEN RETURN; END_IF IF Test_PRG.Swipe_menu = 1 THEN IF Hover_Y < 2 THEN Hover_Y:= Hover_Y + 1; END_IF END_IF IF Test_PRG.Swipe_menu = 0 THEN IF Hover_Y < 5 THEN Hover_Y:= Hover_Y + 1; END_IF END_IF, VisuElemId=-1
    hotkey  Id=481043677184, Key=KeyDown=True, KeyName=right, ActionToExecute=Action=STSnippet=IF xSelected THEN RETURN; END_IF IF Hover_Y > 0 THEN Hover_Y:= Hover_Y - 1; END_IF, VisuElemId=-1
    hotkey  Id=481044725760, Key=KeyDown=True, KeyName=end, ActionToExecute=Action=STSnippet=xSelected:= xSelected XOR TRUE;, VisuElemId=-1
END_VISUALIZATION

// CR1104/Application/HMI/Components/Menu/Menu_Item
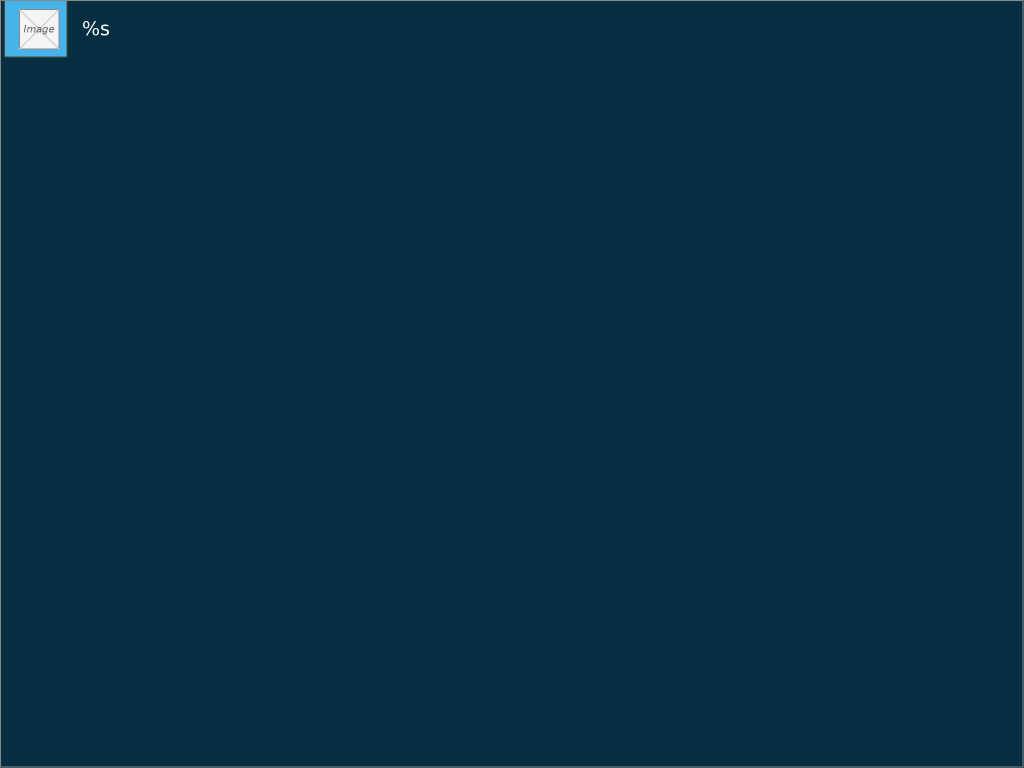
VISUALIZATION Menu_Item  // 1024x768
VAR_INPUT
	_SELECTED: BOOL; 
END_VAR

VAR_INPUT
	Icon: STRING;
	Text: STRING;
	Visu_Reference: STRING;
END_VAR
    RoundedRectangle (4,0 63x57), invisible if: NOT(_SELECTED)
    Image (19,9 40x40)
        p84334746: Icon
    Rectangle (79,1 102x56), "%s", text variable: Text
END_VISUALIZATION

// CR1104/Application/HMI/Components/Menu/Right_Side_Nav
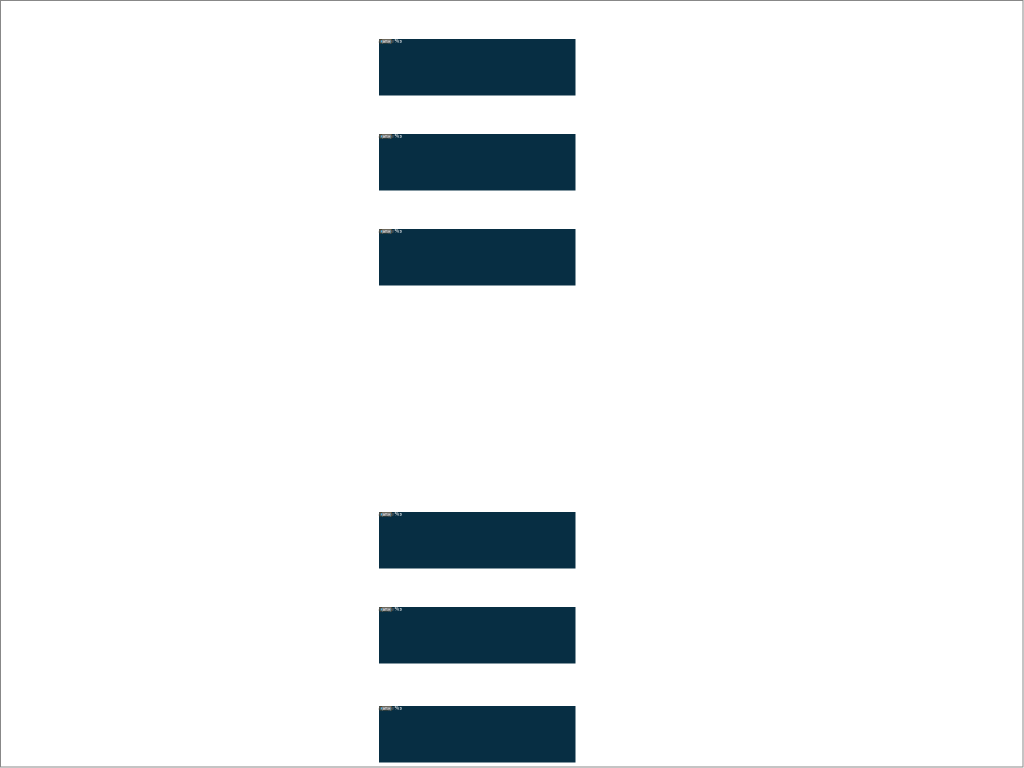
VISUALIZATION Right_Side_Nav  // 1024x768
VAR_INPUT
	Show_Menu: BOOL;
END_VAR


VAR_IN_OUT
	Select_Y: UINT;
END_VAR
    Frame (379,39 196x56)
        shows Menu_Item(_SELECTED := Select_Y = 0, Icon := 'pump_icon', Text := 'Sample')
        pReferences[0]: Key_Reference=0, Icon_selected='pump_3815797'
    Frame (379,134 196x56)
        shows Menu_Item(_SELECTED := Select_Y = 1, Icon := 'pump_icon', Text := 'Sample')
    Frame (379,229 196x56)
        shows Menu_Item(_SELECTED := Select_Y = 2, Icon := 'pump_icon', Text := 'Sample')
    Frame (379,512 196x56)
        shows Menu_Item(_SELECTED := Select_Y = 3, Icon := 'pump_icon', Text := 'Sample')
    Frame (379,607 196x56)
        shows Menu_Item(_SELECTED := Select_Y = 4, Icon := 'pump_icon', Text := 'Sample')
    Frame (379,706 196x56)
        shows Menu_Item(_SELECTED := Select_Y = 5, Icon := 'pump_icon', Text := 'Sample')
    hotkey  Id=481039482880, Key=KeyDown=True, KeyName=left, ActionToExecute=Action=STSnippet=IF NOT(Show_Menu) THEN RETURN; END_IF Select_Y:= Select_Y + 1;, VisuElemId=-1
    hotkey  Id=481040531456, Key=KeyDown=True, KeyName=right, ActionToExecute=Action=STSnippet=IF NOT(Show_Menu) THEN RETURN; END_IF Select_Y:= Select_Y - 1;, VisuElemId=-1
    hotkey  Id=481046822912, Key=KeyDown=True, KeyName=F5, ActionToExecute=Action=STSnippet=Select_Y:= 0;, VisuElemId=-1
    hotkey  Id=481045774336, Key=KeyDown=True, KeyName=F3, ActionToExecute=Action=STSnippet=Select_Y:= 1;, VisuElemId=-1
    hotkey  Id=481044725760, Key=KeyDown=True, KeyName=F1, ActionToExecute=Action=STSnippet=Select_Y:= 2;, VisuElemId=-1
    hotkey  Id=481043677184, Key=KeyDown=True, KeyName=F2, ActionToExecute=Action=STSnippet=Select_Y:= 3;, VisuElemId=-1
    hotkey  Id=481042628608, Key=KeyDown=True, KeyName=F4, ActionToExecute=Action=STSnippet=Select_Y:= 4;, VisuElemId=-1
    hotkey  Id=481041580032, Key=KeyDown=True, KeyName=F6, ActionToExecute=Action=STSnippet=Select_Y:= 5;, VisuElemId=-1
END_VISUALIZATION

// CR1104/Application/HMI/Components/Pages/Analytics
VISUALIZATION Analytics  // 1024x768
END_VISUALIZATION

// CR1104/Application/HMI/Components/Pages/Chemistry
VISUALIZATION Chemistry  // 1024x768
END_VISUALIZATION

// CR1104/Application/HMI/Components/Pages/Overview
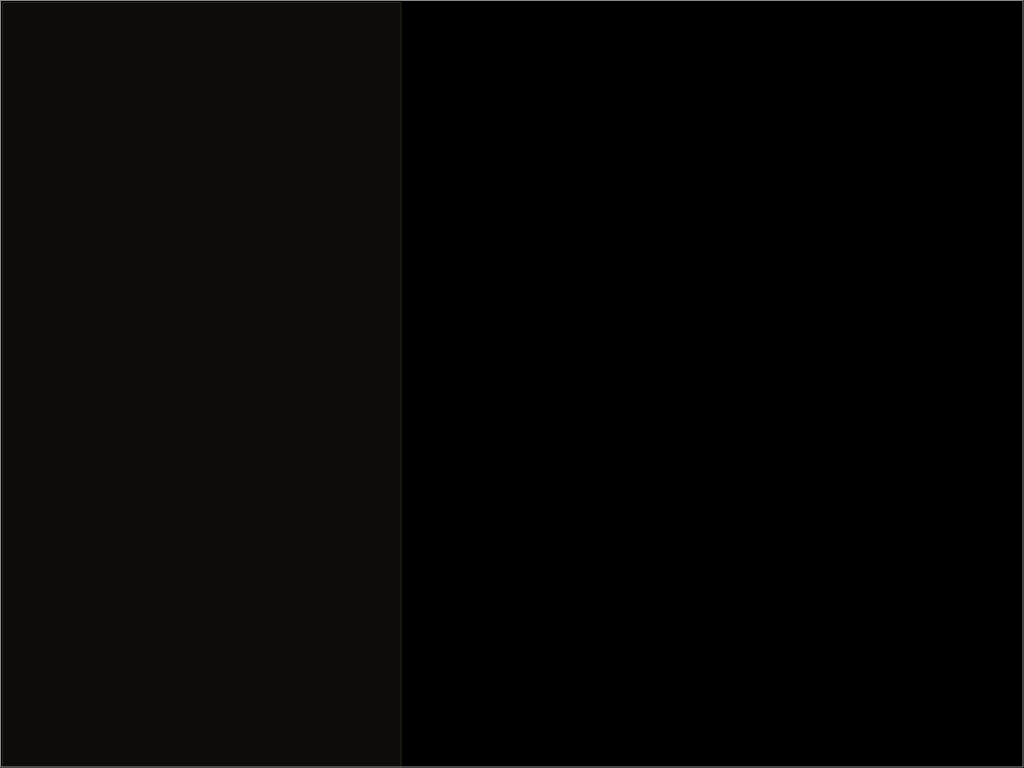
VISUALIZATION Overview  // 1024x768
    RoundedRectangle (2,2 399x794)
END_VISUALIZATION

// CR1104/Application/HMI/Components/Pages/Pumps
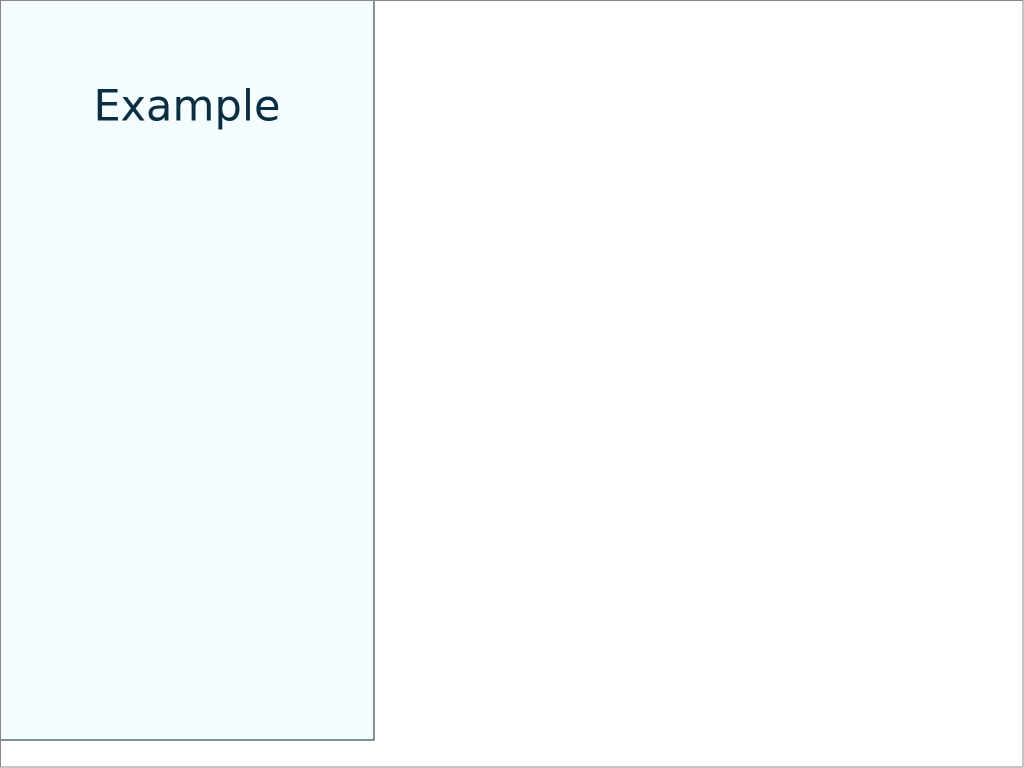
VISUALIZATION Pumps  // 1024x768
    Rectangle (0,0 374x740)
    Rectangle (0,28 374x155), "Example"
END_VISUALIZATION

// CR1104/Application/HMI/Components/Pages/Purge
